Fanuc TP program (LS listing): SET_FRAMES.LS

/PROG  SET_FRAMES
/ATTR
OWNER		= MNEDITOR;
COMMENT		= "";
PROG_SIZE	= 196;
CREATE		= DATE 25-07-22  TIME 10:58:28;
MODIFIED	= DATE 25-07-22  TIME 10:59:30;
FILE_NAME	= ;
VERSION		= 0;
LINE_COUNT	= 4;
MEMORY_SIZE	= 552;
PROTECT		= READ_WRITE;
TCD:  STACK_SIZE	= 0,
      TASK_PRIORITY	= 50,
      TIME_SLICE	= 0,
      BUSY_LAMP_OFF	= 0,
      ABORT_REQUEST	= 0,
      PAUSE_REQUEST	= 0;
DEFAULT_GROUP	= 1,*,*,*,*;
CONTROL_CODE	= 00000000 00000000;
/MN
   1:  UFRAME[6:# Vice1 T1]=PR[1:@ ref vice1 T1] ;
   2:  UFRAME[7:# Vice1 T2]=PR[2:@ ref vice1 T2] ;
   3:  UFRAME[8:# Vice2 T1]=PR[3:@ ref vice2 T1] ;
   4:  UFRAME[9:# Vice2 T2]=PR[4:@ ref vice2 T2] ;
/POS
/END
